// SIMATIC S7-200 project (STEP 7-Micro/WIN), CPU 224 CN REL 02.01

ORGANIZATION_BLOCK 主程序:OB1
TITLE=程序注释
BEGIN
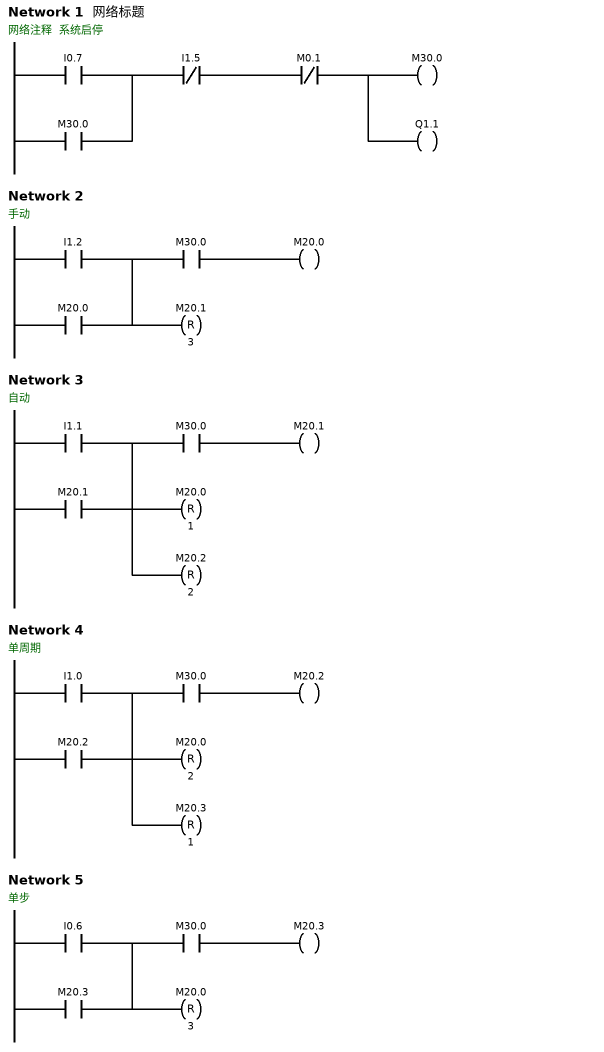
Network 1 // 网络标题
// 网络注释	系统启停
// (network saved uncompiled; LAD cells follow)
// row 0: c0 -| |- I0.7 v  c1 -|/|- I1.5  c2 -|/|- M0.1 v  c3 -( ) M30.0
// row 1: c0 -| |- M30.0 ^  c2 ^  c3 -( ) Q1.1
Network 2
// 手动	
// (network saved uncompiled; LAD cells follow)
// row 0: c0 -| |- I1.2 v  c1 -| |- M30.0  c2 -( ) M20.0
// row 1: c0 -| |- M20.0 ^  c1 -(R) M20.1, 3
Network 3
// 自动
// (network saved uncompiled; LAD cells follow)
// row 0: c0 -| |- I1.1 v  c1 -| |- M30.0  c2 -( ) M20.1
// row 1: c0 -| |- M20.1 ^v  c1 -(R) M20.0, 1
// row 2: c0 ^  c1 -(R) M20.2, 2
Network 4
// 单周期
// (network saved uncompiled; LAD cells follow)
// row 0: c0 -| |- I1.0 v  c1 -| |- M30.0  c2 -( ) M20.2
// row 1: c0 -| |- M20.2 ^v  c1 -(R) M20.0, 2
// row 2: c0 ^  c1 -(R) M20.3, 1
Network 5
// 单步
// (network saved uncompiled; LAD cells follow)
// row 0: c0 -| |- I0.6 v  c1 -| |- M30.0  c2 -( ) M20.3
// row 1: c0 -| |- M20.3 ^  c1 -(R) M20.0, 3
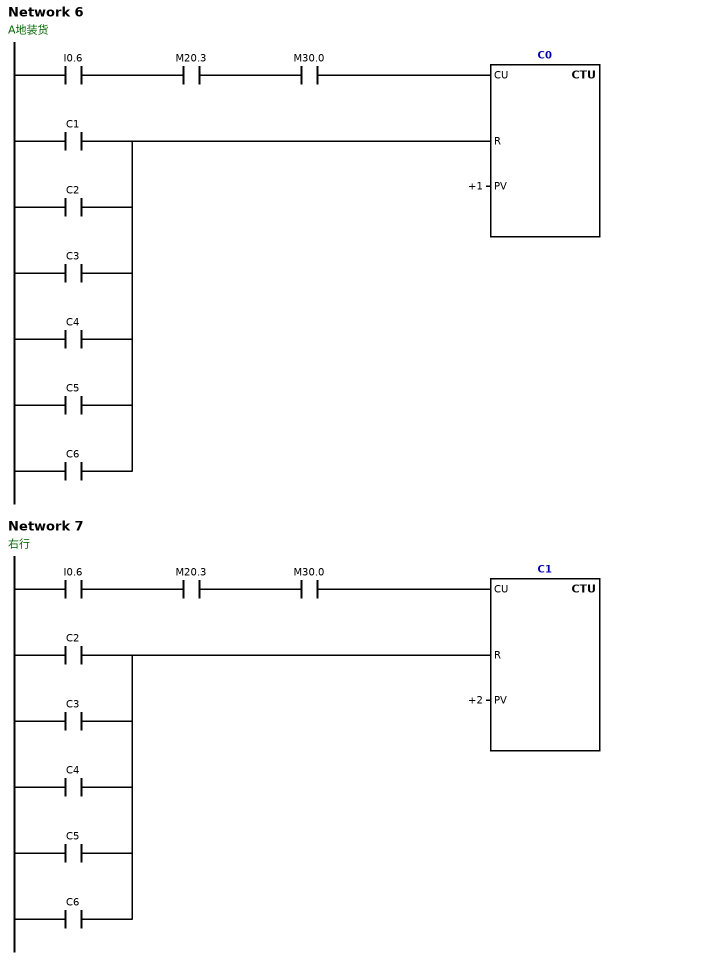
Network 6
// A地装货
// (network saved uncompiled; LAD cells follow)
// row 0: c0 -| |- I0.6  c1 -| |- M20.3  c2 -| |- M30.0  c3 --  c4 [CTU C0 CU:=power@row0, R:=power@row1, PV:=+1]
// row 1: c0 -| |- C1 v  c1 --  c2 --  c3 --  c4 [box]
// row 2: c0 -| |- C2 ^v  c4 [box]
// row 3: c0 -| |- C3 ^v
// row 4: c0 -| |- C4 ^v
// row 5: c0 -| |- C5 ^v
// row 6: c0 -| |- C6 ^
Network 7
// 右行
// (network saved uncompiled; LAD cells follow)
// row 0: c0 -| |- I0.6  c1 -| |- M20.3  c2 -| |- M30.0  c3 --  c4 [CTU C1 CU:=power@row0, R:=power@row1, PV:=+2]
// row 1: c0 -| |- C2 v  c1 --  c2 --  c3 --  c4 [box]
// row 2: c0 -| |- C3 ^v  c4 [box]
// row 3: c0 -| |- C4 ^v
// row 4: c0 -| |- C5 ^v
// row 5: c0 -| |- C6 ^
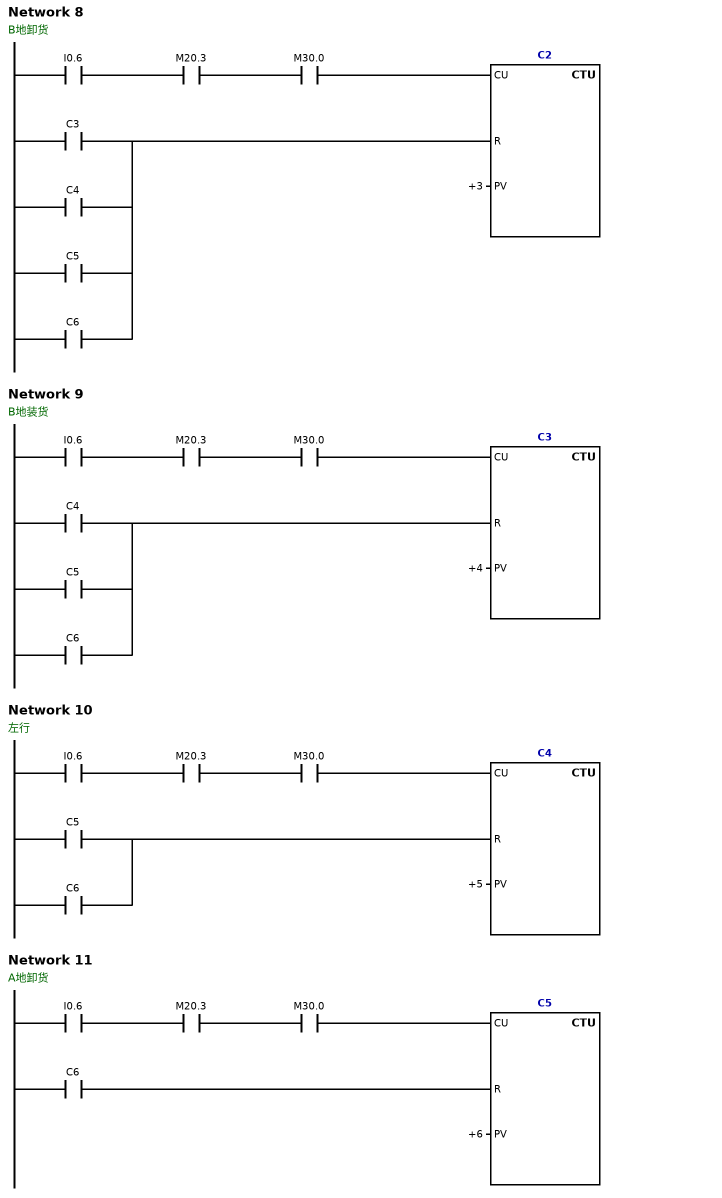
Network 8
// B地卸货
// (network saved uncompiled; LAD cells follow)
// row 0: c0 -| |- I0.6  c1 -| |- M20.3  c2 -| |- M30.0  c3 --  c4 [CTU C2 CU:=power@row0, R:=power@row1, PV:=+3]
// row 1: c0 -| |- C3 v  c1 --  c2 --  c3 --  c4 [box]
// row 2: c0 -| |- C4 ^v  c4 [box]
// row 3: c0 -| |- C5 ^v
// row 4: c0 -| |- C6 ^
Network 9
// B地装货
// (network saved uncompiled; LAD cells follow)
// row 0: c0 -| |- I0.6  c1 -| |- M20.3  c2 -| |- M30.0  c3 --  c4 [CTU C3 CU:=power@row0, R:=power@row1, PV:=+4]
// row 1: c0 -| |- C4 v  c1 --  c2 --  c3 --  c4 [box]
// row 2: c0 -| |- C5 ^v  c4 [box]
// row 3: c0 -| |- C6 ^
Network 10
// 左行
// (network saved uncompiled; LAD cells follow)
// row 0: c0 -| |- I0.6  c1 -| |- M20.3  c2 -| |- M30.0  c3 --  c4 [CTU C4 CU:=power@row0, R:=power@row1, PV:=+5]
// row 1: c0 -| |- C5 v  c1 --  c2 --  c3 --  c4 [box]
// row 2: c0 -| |- C6 ^  c4 [box]
Network 11
// A地卸货
// (network saved uncompiled; LAD cells follow)
// row 0: c0 -| |- I0.6  c1 -| |- M20.3  c2 -| |- M30.0  c3 --  c4 [CTU C5 CU:=power@row0, R:=power@row1, PV:=+6]
// row 1: c0 -| |- C6  c1 --  c2 --  c3 --  c4 [box]
// row 2: c4 [box]
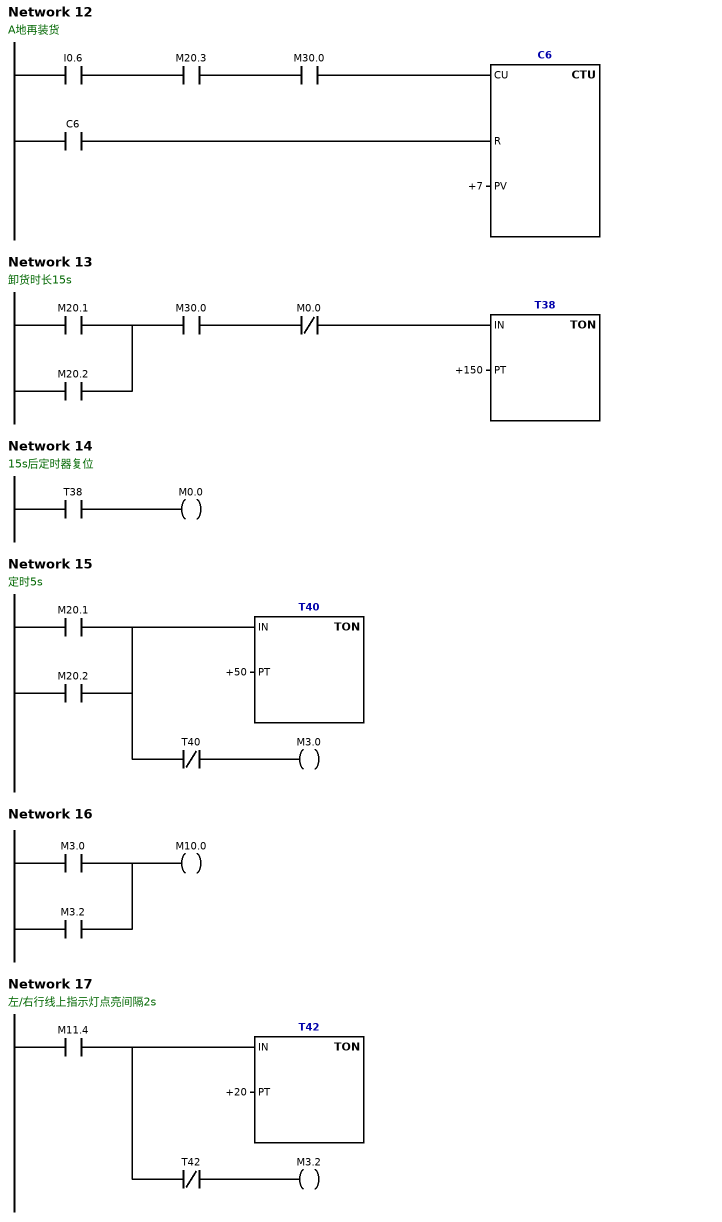
Network 12
// A地再装货
// (network saved uncompiled; LAD cells follow)
// row 0: c0 -| |- I0.6  c1 -| |- M20.3  c2 -| |- M30.0  c3 --  c4 [CTU C6 CU:=power@row0, R:=power@row1, PV:=+7]
// row 1: c0 -| |- C6  c1 --  c2 --  c3 --  c4 [box]
// row 2: c4 [box]
Network 13
// 卸货时长15s
LD     M20.1
O      M20.2
A      M30.0
AN     M0.0
TON    T38, +150
Network 14
// 15s后定时器复位
LD     T38
=      M0.0
Network 15
// 定时5s
LD     M20.1
O      M20.2
TON    T40, +50
AN     T40
=      M3.0
Network 16
LD     M3.0
O      M3.2
=      M10.0
Network 17
// 左/右行线上指示灯点亮间隔2s
LD     M11.4
TON    T42, +20
AN     T42
=      M3.2
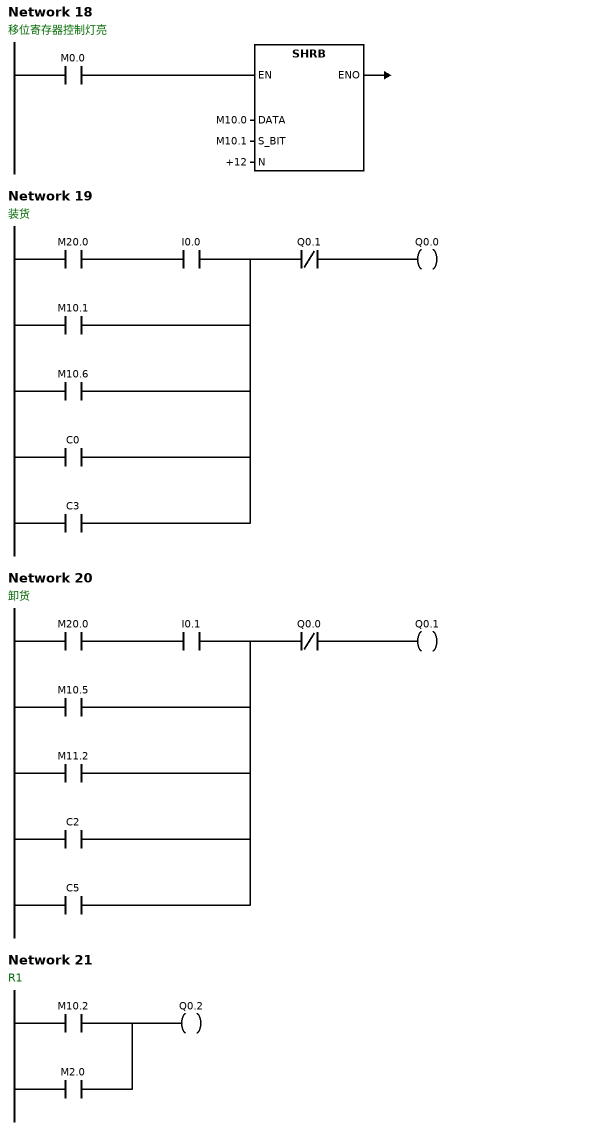
Network 18
// 移位寄存器控制灯亮
LD     M0.0
SHRB   M10.0, M10.1, +12
Network 19
// 装货
// (network saved uncompiled; LAD cells follow)
// row 0: c0 -| |- M20.0  c1 -| |- I0.0 v  c2 -|/|- Q0.1  c3 -( ) Q0.0
// row 1: c0 -| |- M10.1  c1 -- ^v
// row 2: c0 -| |- M10.6  c1 -- ^v
// row 3: c0 -| |- C0  c1 -- ^v
// row 4: c0 -| |- C3  c1 -- ^
Network 20
// 卸货
// (network saved uncompiled; LAD cells follow)
// row 0: c0 -| |- M20.0  c1 -| |- I0.1 v  c2 -|/|- Q0.0  c3 -( ) Q0.1
// row 1: c0 -| |- M10.5  c1 -- ^v
// row 2: c0 -| |- M11.2  c1 -- ^v
// row 3: c0 -| |- C2  c1 -- ^v
// row 4: c0 -| |- C5  c1 -- ^
Network 21
// R1
LD     M10.2
O      M2.0
=      Q0.2
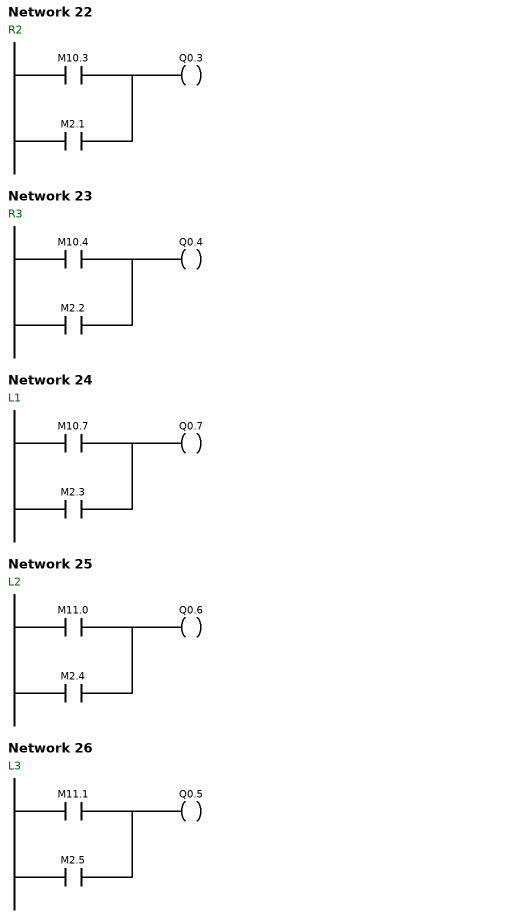
Network 22
// R2
LD     M10.3
O      M2.1
=      Q0.3
Network 23
// R3
LD     M10.4
O      M2.2
=      Q0.4
Network 24
// L1
LD     M10.7
O      M2.3
=      Q0.7
Network 25
// L2
LD     M11.0
O      M2.4
=      Q0.6
Network 26
// L3
LD     M11.1
O      M2.5
=      Q0.5
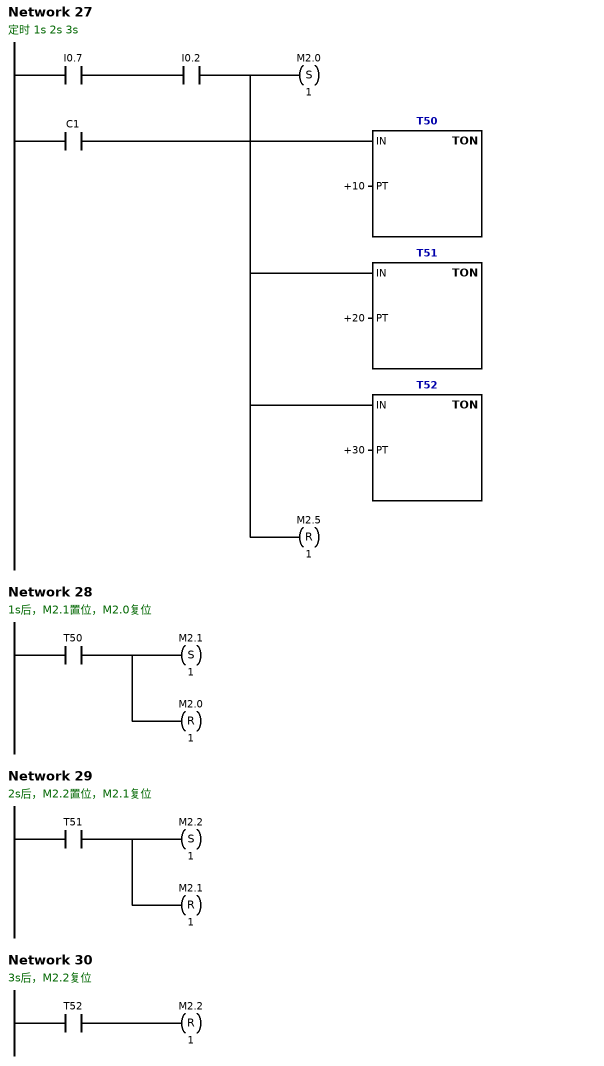
Network 27
// 定时 1s 2s 3s
// (network saved uncompiled; LAD cells follow)
// row 0: c0 -| |- I0.7  c1 -| |- I0.2 v  c2 -(S) M2.0, 1
// row 1: c0 -| |- C1  c1 -- ^v  c2 --  c3 [TON T50 IN:=power@row1, PT:=+10]
// row 2: c1 ^v  c3 [box]
// row 3: c1 ^v  c2 --  c3 [TON T51 IN:=power@row3, PT:=+20]
// row 4: c1 ^v  c3 [box]
// row 5: c1 ^v  c2 --  c3 [TON T52 IN:=power@row5, PT:=+30]
// row 6: c1 ^v  c3 [box]
// row 7: c1 ^  c2 -(R) M2.5, 1
Network 28
// 1s后，M2.1置位，M2.0复位
LD     T50
S      M2.1, 1
R      M2.0, 1
Network 29
// 2s后，M2.2置位，M2.1复位
LD     T51
S      M2.2, 1
R      M2.1, 1
Network 30
// 3s后，M2.2复位
LD     T52
R      M2.2, 1
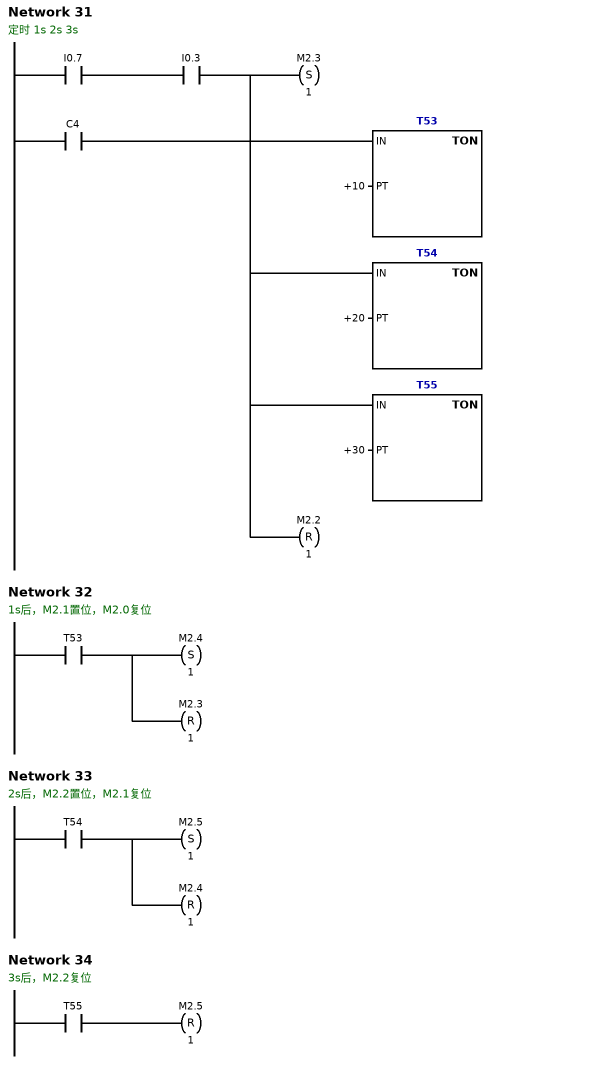
Network 31
// 定时 1s 2s 3s
// (network saved uncompiled; LAD cells follow)
// row 0: c0 -| |- I0.7  c1 -| |- I0.3 v  c2 -(S) M2.3, 1
// row 1: c0 -| |- C4  c1 -- ^v  c2 --  c3 [TON T53 IN:=power@row1, PT:=+10]
// row 2: c1 ^v  c3 [box]
// row 3: c1 ^v  c2 --  c3 [TON T54 IN:=power@row3, PT:=+20]
// row 4: c1 ^v  c3 [box]
// row 5: c1 ^v  c2 --  c3 [TON T55 IN:=power@row5, PT:=+30]
// row 6: c1 ^v  c3 [box]
// row 7: c1 ^  c2 -(R) M2.2, 1
Network 32
// 1s后，M2.1置位，M2.0复位
LD     T53
S      M2.4, 1
R      M2.3, 1
Network 33
// 2s后，M2.2置位，M2.1复位
LD     T54
S      M2.5, 1
R      M2.4, 1
Network 34
// 3s后，M2.2复位
LD     T55
R      M2.5, 1
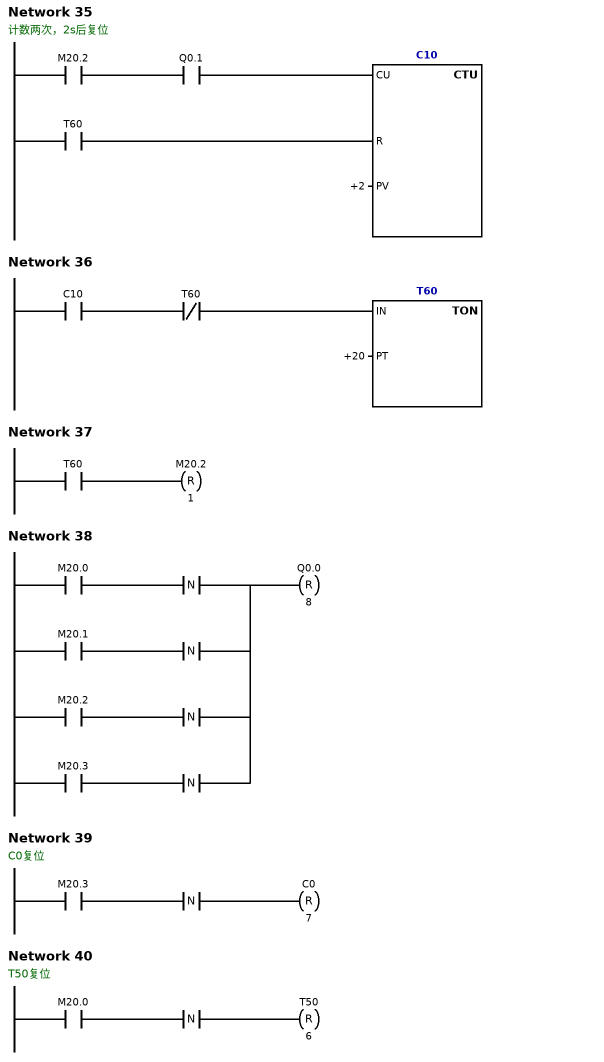
Network 35
// 计数两次，2s后复位
LD     M20.2
A      Q0.1
LD     T60
CTU    C10, +2
Network 36
LD     C10
AN     T60
TON    T60, +20
Network 37
LD     T60
R      M20.2, 1
Network 38
LD     M20.0
ED
LD     M20.1
ED
OLD
LD     M20.2
ED
OLD
LD     M20.3
ED
OLD
R      Q0.0, 8
Network 39
// C0复位
LD     M20.3
ED
R      C0, 7
Network 40
// T50复位
LD     M20.0
ED
R      T50, 6
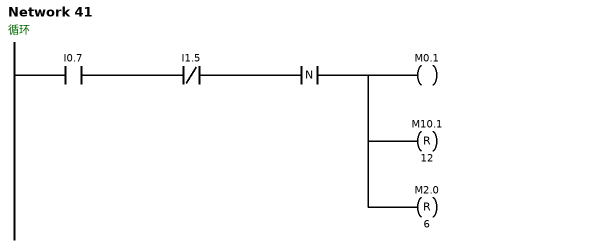
Network 41
// 循环
// (network saved uncompiled; LAD cells follow)
// row 0: c0 -| |- I0.7  c1 -|/|- I1.5  c2 -|N|-  v  c3 -( ) M0.1
// row 1: c2 ^v  c3 -(R) M10.1, 12
// row 2: c2 ^  c3 -(R) M2.0, 6
END_ORGANIZATION_BLOCK
